# EPICS substitutions: bpm_data_combiner_app/Db/bpm_dev_input.substitutions
file "db/bpm_dev_input_rec.db"
{
	pattern { DEV_NAME  }
	        { BPMZ5D8R  }
	        { BPMZ6D8R  }
	        { BPMZ7D8R  }

	        { BPMZ1T8R  }
	        { BPMZ2T8R  }
	        { BPMZ3T8R  }
	        { BPMZ4T8R  }

}
